// Mitsubishi GX Works2 project: water   PLC: FX3U/FX3UC

PROGRAM MAIN
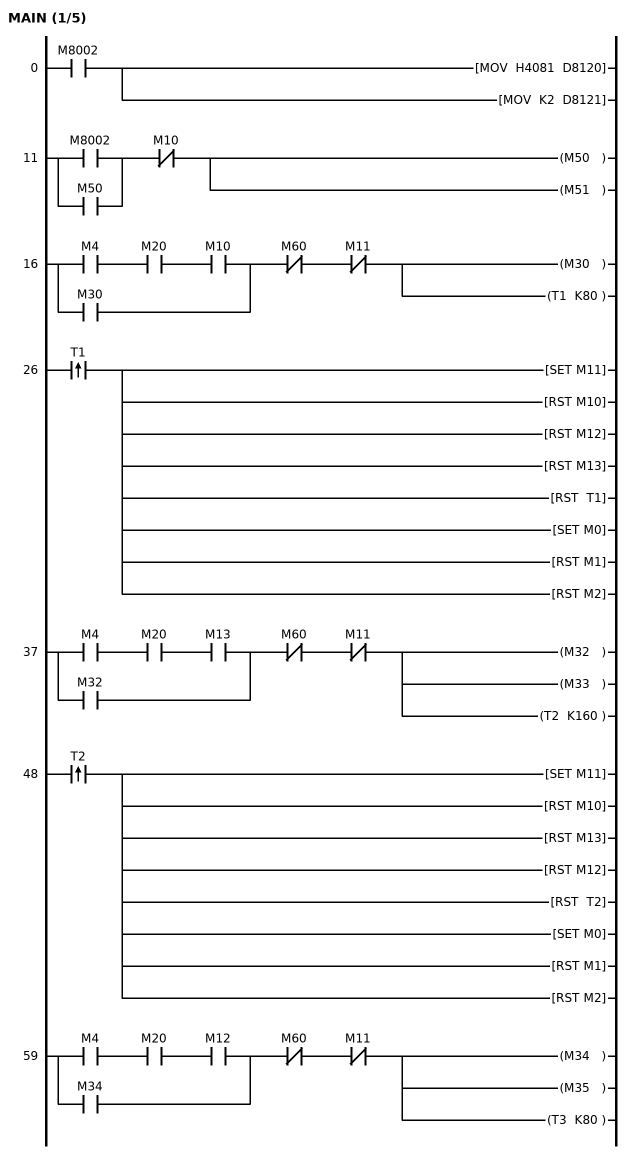
0     LD      M8002
      MOV     H4081 D8120
      MOV     K2 D8121
11    LD      M8002
      OR      M50
      ANI     M10
      OUT     M50
      OUT     M51
16    LD      M4
      AND     M20
      AND     M10
      OR      M30
      ANI     M60
      ANI     M11
      OUT     M30
      OUT     T1 K80
26    LDP     T1
      SET     M11
      RST     M10
      RST     M12
      RST     M13
      RST     T1
      SET     M0
      RST     M1
      RST     M2
37    LD      M4
      AND     M20
      AND     M13
      OR      M32
      ANI     M60
      ANI     M11
      OUT     M32
      OUT     M33
      OUT     T2 K160
48    LDP     T2
      SET     M11
      RST     M10
      RST     M13
      RST     M12
      RST     T2
      SET     M0
      RST     M1
      RST     M2
59    LD      M4
      AND     M20
      AND     M12
      OR      M34
      ANI     M60
      ANI     M11
      OUT     M34
      OUT     M35
      OUT     T3 K80
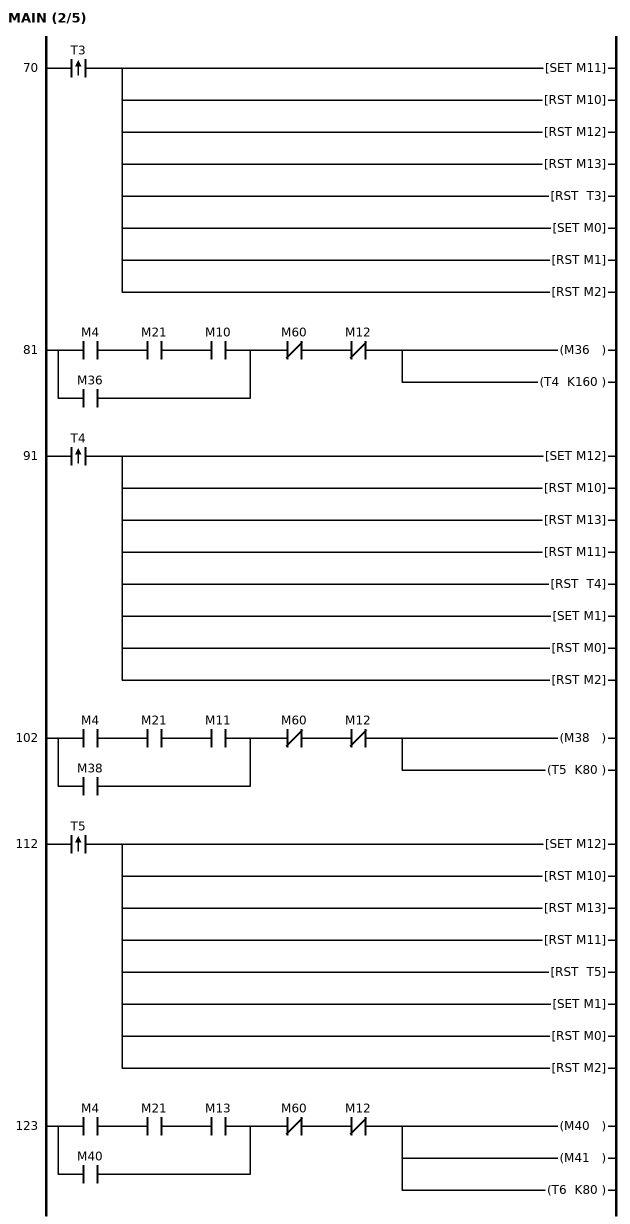
70    LDP     T3
      SET     M11
      RST     M10
      RST     M12
      RST     M13
      RST     T3
      SET     M0
      RST     M1
      RST     M2
81    LD      M4
      AND     M21
      AND     M10
      OR      M36
      ANI     M60
      ANI     M12
      OUT     M36
      OUT     T4 K160
91    LDP     T4
      SET     M12
      RST     M10
      RST     M13
      RST     M11
      RST     T4
      SET     M1
      RST     M0
      RST     M2
102   LD      M4
      AND     M21
      AND     M11
      OR      M38
      ANI     M60
      ANI     M12
      OUT     M38
      OUT     T5 K80
112   LDP     T5
      SET     M12
      RST     M10
      RST     M13
      RST     M11
      RST     T5
      SET     M1
      RST     M0
      RST     M2
123   LD      M4
      AND     M21
      AND     M13
      OR      M40
      ANI     M60
      ANI     M12
      OUT     M40
      OUT     M41
      OUT     T6 K80
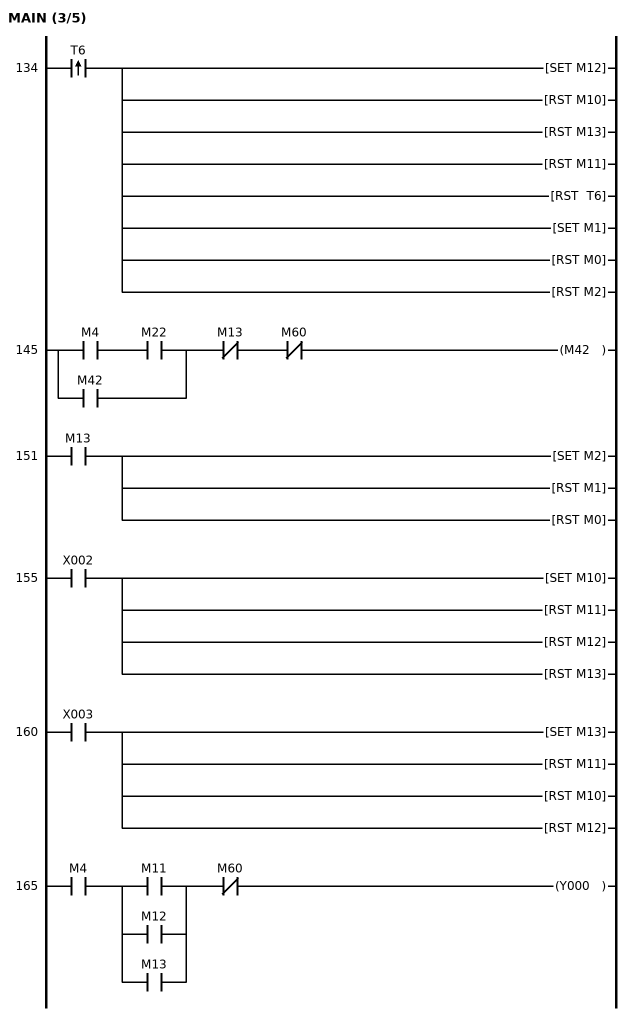
134   LDP     T6
      SET     M12
      RST     M10
      RST     M13
      RST     M11
      RST     T6
      SET     M1
      RST     M0
      RST     M2
145   LD      M4
      AND     M22
      OR      M42
      ANI     M13
      ANI     M60
      OUT     M42
151   LD      M13
      SET     M2
      RST     M1
      RST     M0
155   LD      X002
      SET     M10
      RST     M11
      RST     M12
      RST     M13
160   LD      X003
      SET     M13
      RST     M11
      RST     M10
      RST     M12
165   LD      M4
      LD      M11
      OR      M12
      OR      M13
      ANB
      ANI     M60
      OUT     Y000
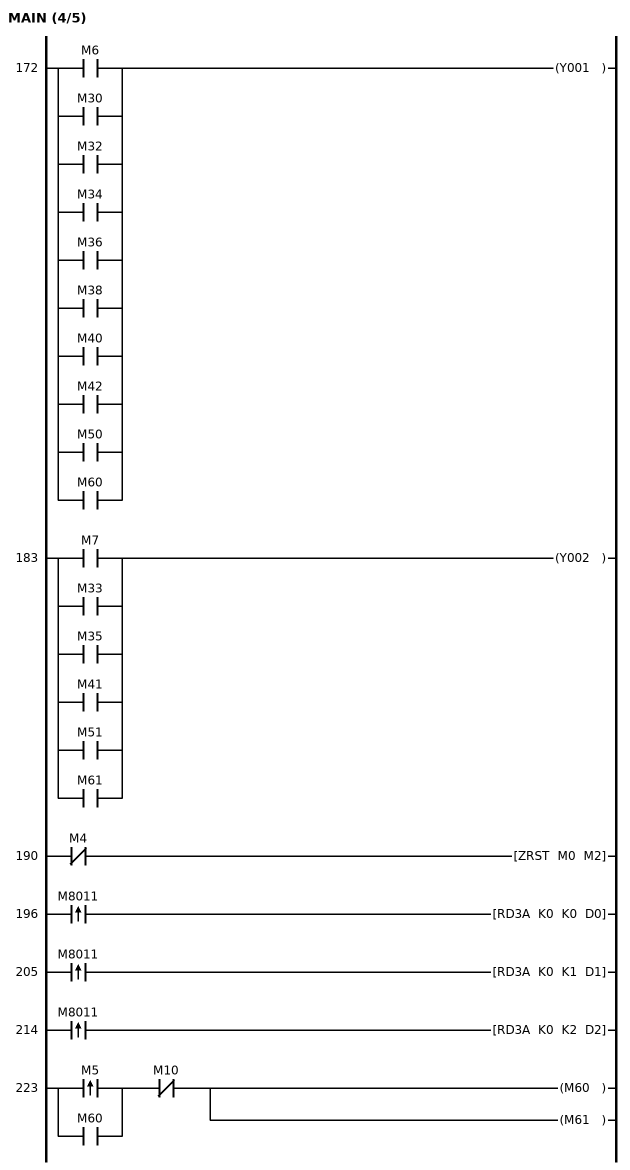
172   LD      M6
      OR      M30
      OR      M32
      OR      M34
      OR      M36
      OR      M38
      OR      M40
      OR      M42
      OR      M50
      OR      M60
      OUT     Y001
183   LD      M7
      OR      M33
      OR      M35
      OR      M41
      OR      M51
      OR      M61
      OUT     Y002
190   LDI     M4
      ZRST    M0 M2
196   LDP     M8011
      RD3A    K0 K0 D0
205   LDP     M8011
      RD3A    K0 K1 D1
214   LDP     M8011
      RD3A    K0 K2 D2
223   LDP     M5
      OR      M60
      ANI     M10
      OUT     M60
      OUT     M61
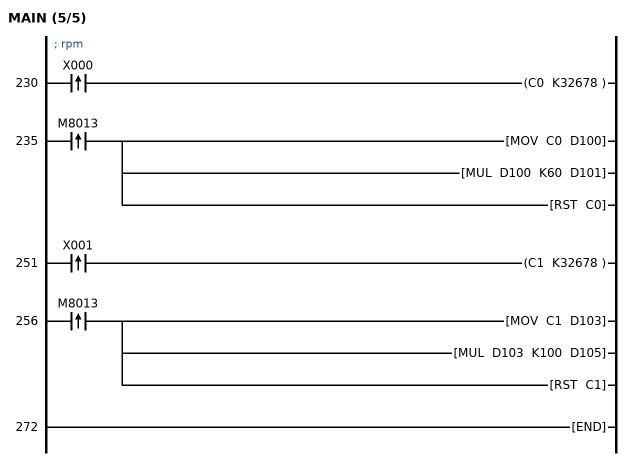
; rpm
230   LDP     X000
      OUT     C0 K32678
235   LDP     M8013
      MOV     C0 D100
      MUL     D100 K60 D101
      RST     C0
251   LDP     X001
      OUT     C1 K32678
256   LDP     M8013
      MOV     C1 D103
      MUL     D103 K100 D105
      RST     C1
272   END
END_PROGRAM

// device comments not shown above
D102  ; rpm
D107  ; flow rate
